Xinje XDPPro project, PLC1: XL3-16 (software 3.7.17c 2024-04-02)

PROGRAM Ladder

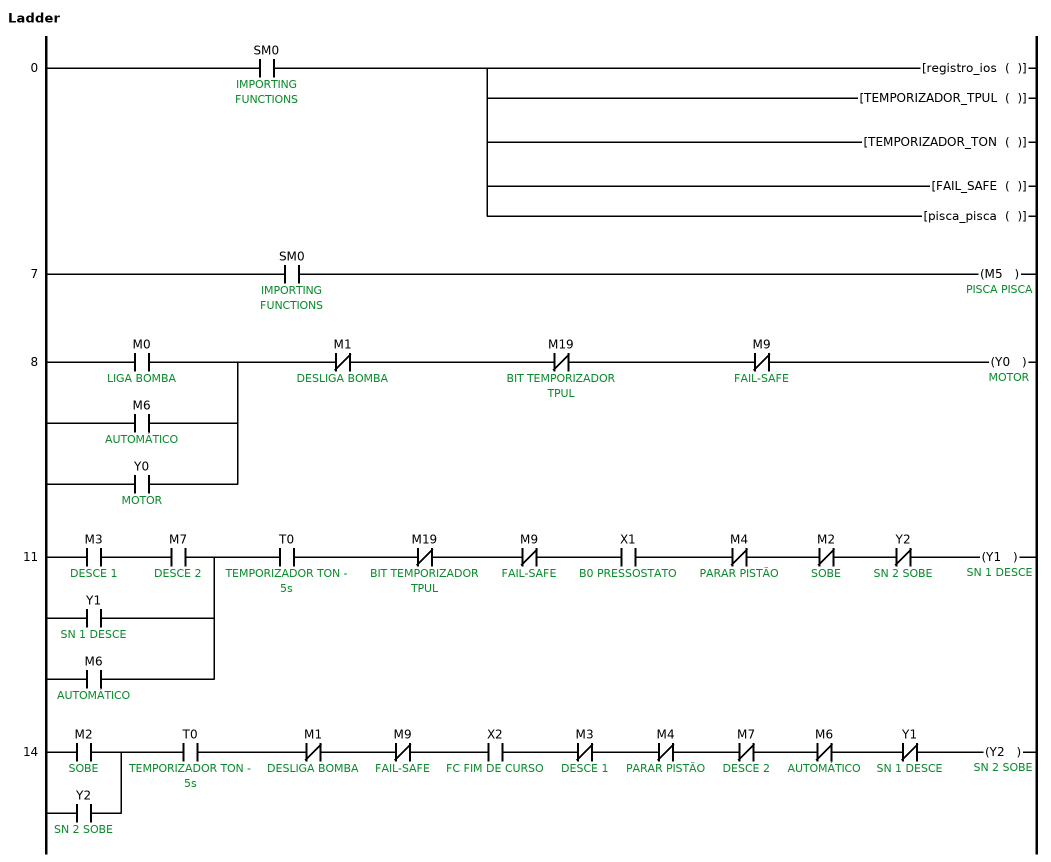
LD     SM0	; IMPORTING FUNCTIONS
registro_ios ( )
TEMPORIZADOR_TPUL ( )
TEMPORIZADOR_TON ( )
FAIL_SAFE ( )
pisca_pisca ( )
LD     SM0	; IMPORTING FUNCTIONS
OUT    M5	; PISCA PISCA
LD     M0	; LIGA BOMBA
OR     M6	; AUTOMÁTICO
OR     Y0	; MOTOR
ANI    M1	; DESLIGA BOMBA
ANI    M19	; BIT TEMPORIZADOR TPUL
ANI    M9	; FAIL-SAFE
OUT    Y0	; MOTOR
LD     M3	; DESCE 1
AND    M7	; DESCE 2
OR     Y1	; SN 1 DESCE
OR     M6	; AUTOMÁTICO
AND    T0	; TEMPORIZADOR TON -  5s
ANI    M19	; BIT TEMPORIZADOR TPUL
ANI    M9	; FAIL-SAFE
AND    X1	; B0 PRESSOSTATO
ANI    M4	; PARAR PISTÃO
ANI    M2	; SOBE
ANI    Y2	; SN 2 SOBE
OUT    Y1	; SN 1 DESCE
LD     M2	; SOBE
OR     Y2	; SN 2 SOBE
AND    T0	; TEMPORIZADOR TON -  5s
ANI    M1	; DESLIGA BOMBA
ANI    M9	; FAIL-SAFE
AND    X2	; FC FIM DE CURSO
ANI    M3	; DESCE 1
ANI    M4	; PARAR PISTÃO
ANI    M7	; DESCE 2
ANI    M6	; AUTOMÁTICO
ANI    Y1	; SN 1 DESCE
OUT    Y2	; SN 2 SOBE

PROGRAM registro_ios

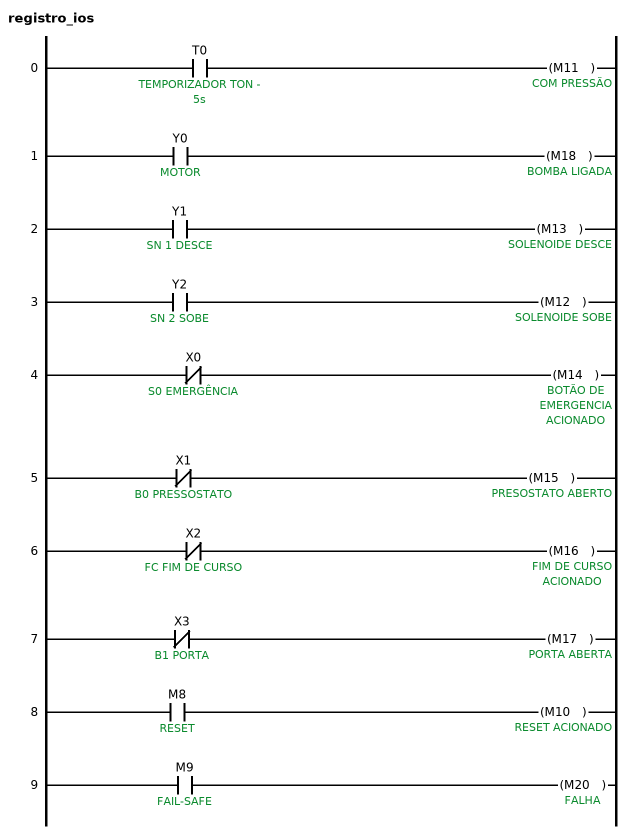
LD     T0	; TEMPORIZADOR TON -  5s
OUT    M11	; COM PRESSÃO
LD     Y0	; MOTOR
OUT    M18	; BOMBA LIGADA
LD     Y1	; SN 1 DESCE
OUT    M13	; SOLENOIDE DESCE
LD     Y2	; SN 2 SOBE
OUT    M12	; SOLENOIDE SOBE
LDI    X0	; S0 EMERGÊNCIA
OUT    M14	; BOTÃO DE EMERGENCIA ACIONADO
LDI    X1	; B0 PRESSOSTATO
OUT    M15	; PRESOSTATO ABERTO
LDI    X2	; FC FIM DE CURSO
OUT    M16	; FIM DE CURSO ACIONADO
LDI    X3	; B1 PORTA
OUT    M17	; PORTA ABERTA
LD     M8	; RESET
OUT    M10	; RESET ACIONADO
LD     M9	; FAIL-SAFE
OUT    M20	; FALHA

PROGRAM TEMPORIZADOR_TPUL

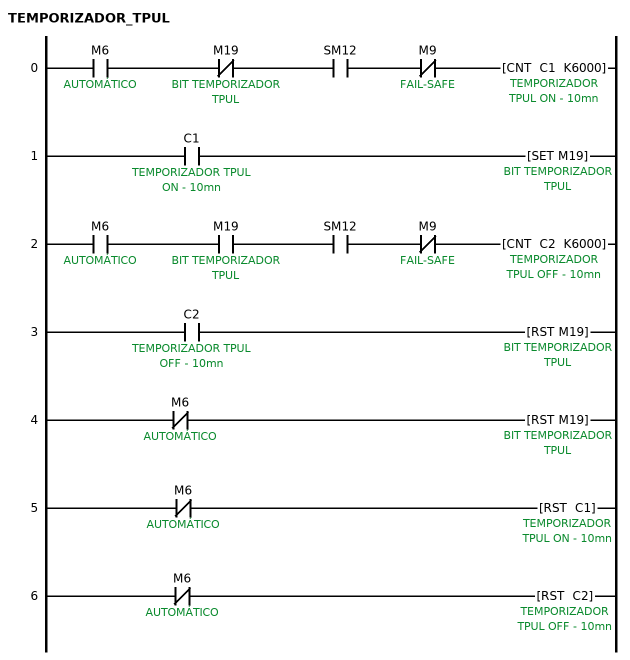
LD     M6	; AUTOMÁTICO
ANI    M19	; BIT TEMPORIZADOR TPUL
AND    SM12
ANI    M9	; FAIL-SAFE
CNT    C1 K6000	; TEMPORIZADOR TPUL ON - 10mn
LD     C1	; TEMPORIZADOR TPUL ON - 10mn
SET    M19	; BIT TEMPORIZADOR TPUL
LD     M6	; AUTOMÁTICO
AND    M19	; BIT TEMPORIZADOR TPUL
AND    SM12
ANI    M9	; FAIL-SAFE
CNT    C2 K6000	; TEMPORIZADOR TPUL OFF - 10mn
LD     C2	; TEMPORIZADOR TPUL OFF - 10mn
RST    M19	; BIT TEMPORIZADOR TPUL
LDI    M6	; AUTOMÁTICO
RST    M19	; BIT TEMPORIZADOR TPUL
LDI    M6	; AUTOMÁTICO
RST    C1	; TEMPORIZADOR TPUL ON - 10mn
LDI    M6	; AUTOMÁTICO
RST    C2	; TEMPORIZADOR TPUL OFF - 10mn

PROGRAM TEMPORIZADOR_TON

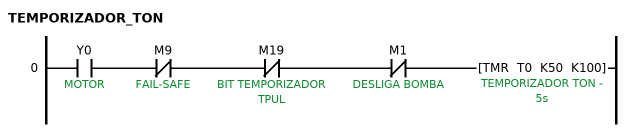
LD     Y0	; MOTOR
ANI    M9	; FAIL-SAFE
ANI    M19	; BIT TEMPORIZADOR TPUL
ANI    M1	; DESLIGA BOMBA
TMR    T0 K50 K100	; TEMPORIZADOR TON -  5s

PROGRAM FAIL_SAFE

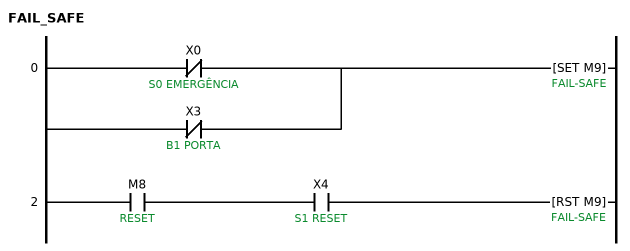
LDI    X0	; S0 EMERGÊNCIA
ORI    X3	; B1 PORTA
SET    M9	; FAIL-SAFE
LD     M8	; RESET
AND    X4	; S1 RESET
RST    M9	; FAIL-SAFE

PROGRAM pisca_pisca

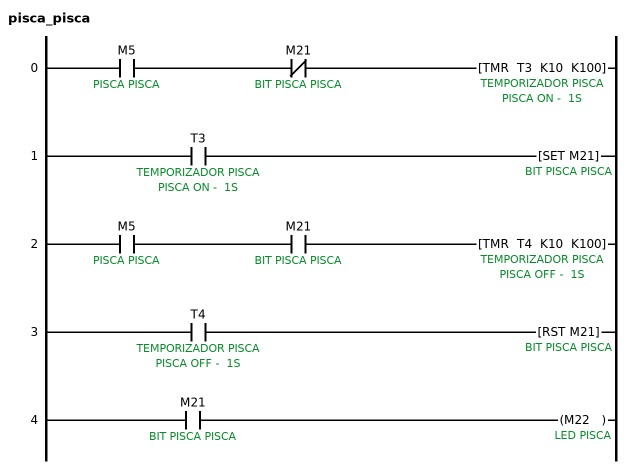
LD     M5	; PISCA PISCA
ANI    M21	; BIT PISCA PISCA
TMR    T3 K10 K100	; TEMPORIZADOR PISCA PISCA ON -  1S
LD     T3	; TEMPORIZADOR PISCA PISCA ON -  1S
SET    M21	; BIT PISCA PISCA
LD     M5	; PISCA PISCA
AND    M21	; BIT PISCA PISCA
TMR    T4 K10 K100	; TEMPORIZADOR PISCA PISCA OFF -  1S
LD     T4	; TEMPORIZADOR PISCA PISCA OFF -  1S
RST    M21	; BIT PISCA PISCA
LD     M21	; BIT PISCA PISCA
OUT    M22	; LED PISCA